{attribute 'GeneratedUsingTerminal: ER1008-0001-0016'}
{attribute addProperty BoxType "ER1008-0001-0016"}
{attribute addProperty Id "InputAT %I*BOOL1"}
{attribute addProperty CRC "2198356929"}
{attribute addProperty Size "1"}
TYPE Channel_830843C1 EXTENDS DigitalInputBase_50022E7B :
STRUCT
	{attribute addProperty Name "Input"}
	Input AT %I* : BOOL;
END_STRUCT
END_TYPE

(* stored: Version 1.2.0.0, ProductVersion 3.1.4024.9
   DUT Channel_830843C1: Id {4919e1d4-ef25-41cb-95c7-69ec792065a1} *)
